DEVICE_TYPE TEST_DEV2 (* Device Type for testing TEST_RES2 *)
  (* Standard: 61499-2 *)
  (* Version 0.1, 2005-05-17, JHC, Holobloc Inc, Changed sockets 1025-6 to 1031-2 to work with WXP. *)
  (* Version 0.0, 2004-06-08, JHC, Rockwell Automation *)
  (* Compiler header: package fb.rt.test; *)
  VAR_INPUT
    INPUT_ID : WSTRING := "225.0.0.1:1031";
    OUTPUT_ID : WSTRING := "225.0.0.1:1032";
  END_VAR
  RESOURCE RES1 : TEST_RES2
  END_RESOURCE
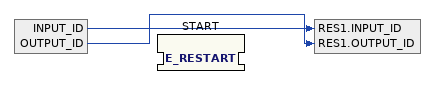
  FBS
    START : E_RESTART;
  END_FBS
  DATA_CONNECTIONS
    INPUT_ID TO RES1.INPUT_ID;
    OUTPUT_ID TO RES1.OUTPUT_ID;
  END_CONNECTIONS
END_DEVICE_TYPE
